FUNCTION_BLOCK PUBLLP0 (* A proxy to 8-Variable local Publisher with interface of global publisher and logic outputs *)
  (* Standard: 61499-2 *)
  (* Version 0.0, 2002-11-12, MLU, VVV *)
  (* Compiler header: package fb.rt.net; *)
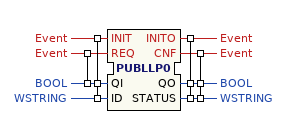
  EVENT_INPUT
    INIT WITH QI, ID; (* Service Initialization *)
    REQ WITH QI; (* Service Request *)
  END_EVENT
  EVENT_OUTPUT
    INITO WITH QO, STATUS; (* Initialization Confirm *)
    CNF WITH QO, STATUS; (* Service Confirmation *)
  END_EVENT
  VAR_INPUT
    QI : BOOL; (* Event Input Qualifier *)
    ID : WSTRING; (* Connection Identifier *)
  END_VAR
  VAR_OUTPUT
    QO : BOOL; (* Event Output Qualifier *)
    STATUS : WSTRING; (* Service Status *)
  END_VAR
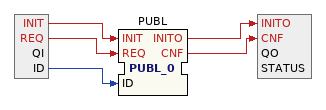
  FBS
    PUBL : PUBL_0;
  END_FBS
  EVENT_CONNECTIONS
    INIT TO PUBL.INIT;
    REQ TO PUBL.REQ;
    PUBL.INITO TO INITO;
    PUBL.CNF TO CNF;
  END_CONNECTIONS
  DATA_CONNECTIONS
    ID TO PUBL.ID;
  END_CONNECTIONS
END_FUNCTION_BLOCK
